FUNCTION F_SafeTo_UDINT : UDINT
VAR_INPUT
	nCovertVar	: Dint;
END_VAR
VAR
END_VAR

F_SafeTo_UDINT := TO_UDINT(MAX(0,nCovertVar));

END_FUNCTION

(* stored: Version 1.1.0.1
   POU F_SafeTo_UDINT: Id {e57ec556-65f3-432c-b1d6-e2eb11108bee}, SpecialFunc None *)
